PROGRAM SafetyInterface_MtrCntrl052
VAR
	
	pMtrRunning: POINTER TO ConvMtrRunningPuck;
	pSafety: POINTER TO Plc2PlcDataSafetyPuckConv;
	
// Stn052_05_StnMain.MotorCtrl
// Call to motor control function block for each main line motor
// Blue Recv - Enc54: 7, 8, 9  Enc55: 5,6
// Red Recv  - Enc54: 4, 5, 6  Enc55: 3, 4
// Grn Recv  - Enc54: 1, 2, 3  Enc55: 1, 2

	{attribute 'TcLinkToOSO':= '	
		.Enc055Mtr01.iDisconnectOk :=  <0,1,4>TIIB[N31S00 (AL1332)]^N31S05 (AL2341)^TxPDO^input byte 1;
		.Enc055Mtr02.iDisconnectOk :=  <0,1,2>TIIB[N32S00 (AL1332)]^N32S01 (AL2341)^TxPDO^input byte 3;
		.Enc055Mtr03.iDisconnectOk :=  <0,1,4>TIIB[N31S00 (AL1332)]^N31S07 (AL2341)^TxPDO^input byte 3;
		.Enc055Mtr04.iDisconnectOk :=  <0,1,3>TIIB[N32S00 (AL1332)]^N32S01 (AL2341)^TxPDO^input byte 1;
		.Enc055Mtr05.iDisconnectOk :=  <0,1,4>TIIB[N31S00 (AL1332)]^N31S05 (AL2341)^TxPDO^input byte 3;
		.Enc055Mtr06.iDisconnectOk :=  <0,1,3>TIIB[N32S00 (AL1332)]^N32S01 (AL2341)^TxPDO^input byte 3;
		.Enc054Mtr01.iDisconnectOk :=  <0,1,3>TIIB[N26S00 (AL1332)]^N26S04 (AL2341)^TxPDO^input byte 3;
		.Enc054Mtr02.iDisconnectOk :=  <0,1,3>TIIB[N27S00 (AL1332)]^N27S04 (AL2341)^TxPDO^input byte 3;
		.Enc054Mtr03.iDisconnectOk :=  <0,1,3>TIIB[N27S00 (AL1332)]^N27S04 (AL2341)^TxPDO^input byte 3;
		.Enc054Mtr04.iDisconnectOk :=  <0,1,4>TIIB[N26S00 (AL1332)]^N26S04 (AL2341)^TxPDO^input byte 1;
		.Enc054Mtr05.iDisconnectOk :=  <0,1,4>TIIB[N27S00 (AL1332)]^N27S04 (AL2341)^TxPDO^input byte 1;
		.Enc054Mtr06.iDisconnectOk :=  <0,1,4>TIIB[N28S00 (AL1332)]^N28S04 (AL2341)^TxPDO^input byte 1;
		.Enc054Mtr07.iDisconnectOk :=  <0,1,4>TIIB[N26S00 (AL1332)]^N26S04 (AL2341)^TxPDO^input byte 3;
		.Enc054Mtr08.iDisconnectOk :=  <0,1,4>TIIB[N27S00 (AL1332)]^N27S04 (AL2341)^TxPDO^input byte 3;
		.Enc054Mtr09.iDisconnectOk :=  <0,1,4>TIIB[N28S00 (AL1332)]^N28S04 (AL2341)^TxPDO^input byte 3'}
	{attribute 'TcLinkTo':= '	
		.Enc055Mtr01.iOverloadTripped := TIIB[N30S06 (EL1008)]^Channel 6^Input;
		.Enc055Mtr02.iOverloadTripped := TIIB[N30S06 (EL1008)]^Channel 8^Input;
		.Enc055Mtr03.iOverloadTripped := TIIB[N30S07 (EL1008)]^Channel 2^Input;
		.Enc055Mtr04.iOverloadTripped := TIIB[N30S07 (EL1008)]^Channel 4^Input;
		.Enc055Mtr05.iOverloadTripped := TIIB[N30S07 (EL1008)]^Channel 6^Input;
		.Enc055Mtr06.iOverloadTripped := TIIB[N30S07 (EL1008)]^Channel 8^Input;
		.Enc054Mtr01.iOverloadTripped := TIIB[N25S06 (EL1008)]^Channel 6^Input;
		.Enc054Mtr02.iOverloadTripped := TIIB[N25S06 (EL1008)]^Channel 8^Input;
		.Enc054Mtr03.iOverloadTripped := TIIB[N25S07 (EL1008)]^Channel 2^Input;
		.Enc054Mtr04.iOverloadTripped := TIIB[N25S07 (EL1008)]^Channel 4^Input;
		.Enc054Mtr05.iOverloadTripped := TIIB[N25S07 (EL1008)]^Channel 6^Input;
		.Enc054Mtr06.iOverloadTripped := TIIB[N25S07 (EL1008)]^Channel 8^Input;
		.Enc054Mtr07.iOverloadTripped := TIIB[N25S08 (EL1008)]^Channel 2^Input;
		.Enc054Mtr08.iOverloadTripped := TIIB[N25S08 (EL1008)]^Channel 4^Input;
		.Enc054Mtr09.iOverloadTripped := TIIB[N25S08 (EL1008)]^Channel 6^Input;
		.Enc055Mtr01.iRunning := TIIB[N30S06 (EL1008)]^Channel 5^Input;
		.Enc055Mtr02.iRunning := TIIB[N30S06 (EL1008)]^Channel 7^Input;
		.Enc055Mtr03.iRunning := TIIB[N30S07 (EL1008)]^Channel 1^Input;
		.Enc055Mtr04.iRunning := TIIB[N30S07 (EL1008)]^Channel 3^Input;
		.Enc055Mtr05.iRunning := TIIB[N30S07 (EL1008)]^Channel 5^Input;
		.Enc055Mtr06.iRunning := TIIB[N30S07 (EL1008)]^Channel 7^Input;
		.Enc054Mtr01.iRunning := TIIB[N25S06 (EL1008)]^Channel 5^Input;
		.Enc054Mtr02.iRunning := TIIB[N25S06 (EL1008)]^Channel 7^Input;
		.Enc054Mtr03.iRunning := TIIB[N25S07 (EL1008)]^Channel 1^Input;
		.Enc054Mtr04.iRunning := TIIB[N25S07 (EL1008)]^Channel 3^Input;
		.Enc054Mtr05.iRunning := TIIB[N25S07 (EL1008)]^Channel 5^Input;
		.Enc054Mtr06.iRunning := TIIB[N25S07 (EL1008)]^Channel 7^Input;
		.Enc054Mtr07.iRunning := TIIB[N25S08 (EL1008)]^Channel 1^Input;
		.Enc054Mtr08.iRunning := TIIB[N25S08 (EL1008)]^Channel 3^Input;
		.Enc054Mtr09.iRunning := TIIB[N25S08 (EL1008)]^Channel 5^Input;
		.Enc055Mtr01.oRun := TIIB[N30S12 (EL2008)]^Channel 4^Output;
		.Enc055Mtr02.oRun := TIIB[N30S12 (EL2008)]^Channel 5^Output;
		.Enc055Mtr03.oRun := TIIB[N30S12 (EL2008)]^Channel 6^Output;
		.Enc055Mtr04.oRun := TIIB[N30S12 (EL2008)]^Channel 7^Output;
		.Enc055Mtr05.oRun := TIIB[N30S12 (EL2008)]^Channel 8^Output;
		.Enc055Mtr06.oRun := TIIB[N30S13 (EL2008)]^Channel 1^Output;
		.Enc054Mtr01.oRun := TIIB[N25S12 (EL2008)]^Channel 5^Output;
		.Enc054Mtr02.oRun := TIIB[N25S12 (EL2008)]^Channel 6^Output;
		.Enc054Mtr03.oRun := TIIB[N25S12 (EL2008)]^Channel 7^Output;
		.Enc054Mtr04.oRun := TIIB[N25S12 (EL2008)]^Channel 8^Output;
		.Enc054Mtr05.oRun := TIIB[N25S13 (EL2008)]^Channel 1^Output;
		.Enc054Mtr06.oRun := TIIB[N25S13 (EL2008)]^Channel 2^Output;
		.Enc054Mtr07.oRun := TIIB[N25S13 (EL2008)]^Channel 3^Output;
		.Enc054Mtr08.oRun := TIIB[N25S13 (EL2008)]^Channel 4^Output;
		.Enc054Mtr09.oRun := TIIB[N25S13 (EL2008)]^Channel 5^Output'}
	MtrCtrls: ConvMtrCtrlsPuck;

	MtrNOKtoRun : BOOL;	
	cntMotorStartIndex: DINT;	
	tmrMotorStartIndex: TON;


END_VAR
VAR CONSTANT	
	
	cMaxMotorStartIndex :DINT := 9;  //If starting pairs of motors  adjust to max number of motors "per enclosure" /2
	
END_VAR

pMtrRunning := ADR(gProduced_SafetyInterfaceConv.MtrRunning);
pSafety := ADR(gProduced_SafetyInterfaceConv);

//Create sequenced motor start index - to prevent inrush overloads at time of motor start		
tmrMotorStartIndex(IN:=NOT tmrMotorStartIndex.Q,PT:=T#300ms);		
IF tmrMotorStartIndex.Q THEN 		
	cntMotorStartIndex := cntMotorStartIndex + 1;	
	IF cntMotorStartIndex > cMaxMotorStartIndex THEN 	
		cntMotorStartIndex := 1;
	END_IF	
END_IF		

// Call action code block that does call for each main line motor		
MotorCtrl();

//distibute the incoming stn data (consumed data from stn) to single produced outgoing to all stns
//MEMCPY(ADR(gProduced_SafetyInterfaceConv.gMtrRunningStn051), ADR(gMtrRunning), SizeOf(gProduced_SafetyInterfaceConv.gMtrRunningStn051));

ACTION MotorCtrl:
// Stn052_05_StnMain.MotorCtrl
// Call to motor control function block for each main line motor
// Blue Recv - Enc54: 7, 8, 9  Enc55: 5,6
// Red Recv  - Enc54: 4, 5, 6  Enc55: 3, 4
// Grn Recv  - Enc54: 1, 2, 3  Enc55: 1, 2
MtrCtrls.Enc054Mtr01(
	CycleAuto := gConsumed_Stn052ToSafetyInterface.CycleAuto,
	CycleReset := gConsumed_Stn052ToSafetyInterface.CycleReset,
	NOKtoRun := pSafety^.Enc054.iEstopRlyTripped,	
//	NOKtoRun := pSafety^.Enc054.iEstopRlyTripped OR 
//		NOT gConsumed_Stn052ToSafetyInterface.Stn052PLCData[2].3 OR 
//		NOT gConsumed_Stn052ToSafetyInterface_OK,		
	StartIndexThisMotor := 1,
	StartIndexCurrent := cntMotorStartIndex,
	hoMtrName := 'Enc054-Mtr1',
	MtrRunning => pMtrRunning^.Enc054Mtr01);

MtrCtrls.Enc054Mtr02(	
	CycleAuto := gConsumed_Stn052ToSafetyInterface.CycleAuto,
	CycleReset := gConsumed_Stn052ToSafetyInterface.CycleReset,
	NOKtoRun := pSafety^.Enc054.iEstopRlyTripped,	
//	NOKtoRun := pSafety^.Enc054.iEstopRlyTripped OR 
//		NOT gConsumed_Stn052ToSafetyInterface.Stn052PLCData[2].3 OR 
//		NOT gConsumed_Stn052ToSafetyInterface_OK,		
	StartIndexThisMotor := 1,
	StartIndexCurrent := cntMotorStartIndex,
	hoMtrName := 'Enc054-Mtr2',
	MtrRunning => pMtrRunning^.Enc054Mtr02);

MtrCtrls.Enc054Mtr03(	
	CycleAuto := gConsumed_Stn052ToSafetyInterface.CycleAuto,
	CycleReset := gConsumed_Stn052ToSafetyInterface.CycleReset,
	NOKtoRun := pSafety^.Enc054.iEstopRlyTripped,	
//	NOKtoRun := pSafety^.Enc054.iEstopRlyTripped OR 
//		NOT gConsumed_Stn052ToSafetyInterface.Stn052PLCData[2].3 OR 
//		NOT gConsumed_Stn052ToSafetyInterface_OK,		
	StartIndexThisMotor := 2,
	StartIndexCurrent := cntMotorStartIndex,
	hoMtrName := 'Enc054-Mtr3',
	MtrRunning => pMtrRunning^.Enc054Mtr03);

MtrCtrls.Enc054Mtr04(	
	CycleAuto := gConsumed_Stn052ToSafetyInterface.CycleAuto,
	CycleReset := gConsumed_Stn052ToSafetyInterface.CycleReset,
	NOKtoRun := pSafety^.Enc054.iEstopRlyTripped,	
//	NOKtoRun := pSafety^.Enc054.iEstopRlyTripped OR 
//		NOT gConsumed_Stn052ToSafetyInterface.Stn052PLCData[2].3 OR 
//		NOT gConsumed_Stn052ToSafetyInterface_OK,		
	StartIndexThisMotor := 2,
	StartIndexCurrent := cntMotorStartIndex,
	hoMtrName := 'Enc054-Mtr4',
	MtrRunning => pMtrRunning^.Enc054Mtr04);

MtrCtrls.Enc054Mtr05(	
	CycleAuto := gConsumed_Stn052ToSafetyInterface.CycleAuto,
	CycleReset := gConsumed_Stn052ToSafetyInterface.CycleReset,
	NOKtoRun := pSafety^.Enc054.iEstopRlyTripped,	
//	NOKtoRun := pSafety^.Enc054.iEstopRlyTripped OR 
//		NOT gConsumed_Stn052ToSafetyInterface.Stn052PLCData[2].3 OR 
//		NOT gConsumed_Stn052ToSafetyInterface_OK,		
	StartIndexThisMotor := 3,
	StartIndexCurrent := cntMotorStartIndex,
	hoMtrName := 'Enc054-Mtr5',
	MtrRunning => pMtrRunning^.Enc054Mtr05);

MtrCtrls.Enc054Mtr06(	
	CycleAuto := gConsumed_Stn052ToSafetyInterface.CycleAuto,
	CycleReset := gConsumed_Stn052ToSafetyInterface.CycleReset,
	NOKtoRun := pSafety^.Enc054.iEstopRlyTripped,	
//	NOKtoRun := pSafety^.Enc054.iEstopRlyTripped OR 
//		NOT gConsumed_Stn052ToSafetyInterface.Stn052PLCData[2].3 OR 
//		NOT gConsumed_Stn052ToSafetyInterface_OK,		
	StartIndexThisMotor := 3,
	StartIndexCurrent := cntMotorStartIndex,
	hoMtrName := 'Enc054-Mtr6',
	MtrRunning => pMtrRunning^.Enc054Mtr06);

MtrCtrls.Enc054Mtr07(	
	CycleAuto := gConsumed_Stn052ToSafetyInterface.CycleAuto,
	CycleReset := gConsumed_Stn052ToSafetyInterface.CycleReset,
	NOKtoRun := pSafety^.Enc054.iEstopRlyTripped,	
//	NOKtoRun := pSafety^.Enc054.iEstopRlyTripped OR 
//		NOT gConsumed_Stn052ToSafetyInterface.Stn052PLCData[2].3 OR 
//		NOT gConsumed_Stn052ToSafetyInterface_OK,		
	StartIndexThisMotor := 4,
	StartIndexCurrent := cntMotorStartIndex,
	hoMtrName := 'Enc054-Mtr7',
	MtrRunning => pMtrRunning^.Enc054Mtr07);

MtrCtrls.Enc054Mtr08(	
	CycleAuto := gConsumed_Stn052ToSafetyInterface.CycleAuto,
	CycleReset := gConsumed_Stn052ToSafetyInterface.CycleReset,
	NOKtoRun := pSafety^.Enc054.iEstopRlyTripped,	
//	NOKtoRun := pSafety^.Enc054.iEstopRlyTripped OR 
//		NOT gConsumed_Stn052ToSafetyInterface.Stn052PLCData[2].3 OR 
//		NOT gConsumed_Stn052ToSafetyInterface_OK,		
	StartIndexThisMotor := 4,
	StartIndexCurrent := cntMotorStartIndex,
	hoMtrName := 'Enc054-Mtr8',
	MtrRunning => pMtrRunning^.Enc054Mtr08);

MtrCtrls.Enc054Mtr09(	
	CycleAuto := gConsumed_Stn052ToSafetyInterface.CycleAuto,
	CycleReset := gConsumed_Stn052ToSafetyInterface.CycleReset,
	NOKtoRun := pSafety^.Enc054.iEstopRlyTripped,	
//	NOKtoRun := pSafety^.Enc054.iEstopRlyTripped OR 
//		NOT gConsumed_Stn052ToSafetyInterface.Stn052PLCData[2].3 OR 
//		NOT gConsumed_Stn052ToSafetyInterface_OK,		
	StartIndexThisMotor := 5,
	StartIndexCurrent := cntMotorStartIndex,
	hoMtrName := 'Enc054-Mtr9',
	MtrRunning => pMtrRunning^.Enc054Mtr09);

MtrCtrls.Enc055Mtr01(	
	CycleAuto := gConsumed_Stn052ToSafetyInterface.CycleAuto,
	CycleReset := gConsumed_Stn052ToSafetyInterface.CycleReset,
	NOKtoRun := pSafety^.Enc055.iEstopRlyTripped,	
//	NOKtoRun := pSafety^.Enc055.iEstopRlyTripped OR 
//		NOT gConsumed_Stn052ToSafetyInterface.Stn052PLCData[2].3 OR 
//		NOT gConsumed_Stn052ToSafetyInterface_OK,		
	StartIndexThisMotor := 1,
	StartIndexCurrent := cntMotorStartIndex,
	hoMtrName := 'Enc055-Mtr1',
	MtrRunning => pMtrRunning^.Enc055Mtr01);

MtrCtrls.Enc055Mtr02(	
	CycleAuto := gConsumed_Stn052ToSafetyInterface.CycleAuto,
	CycleReset := gConsumed_Stn052ToSafetyInterface.CycleReset,
	NOKtoRun := pSafety^.Enc055.iEstopRlyTripped,	
//	NOKtoRun := pSafety^.Enc055.iEstopRlyTripped OR 
//		NOT gConsumed_Stn052ToSafetyInterface.Stn052PLCData[2].3 OR 
//		NOT gConsumed_Stn052ToSafetyInterface_OK,		
	StartIndexThisMotor := 1,
	StartIndexCurrent := cntMotorStartIndex,
	hoMtrName := 'Enc055-Mtr2',
	MtrRunning => pMtrRunning^.Enc055Mtr02);

MtrCtrls.Enc055Mtr03(	
	CycleAuto := gConsumed_Stn052ToSafetyInterface.CycleAuto,
	CycleReset := gConsumed_Stn052ToSafetyInterface.CycleReset,
	NOKtoRun := pSafety^.Enc055.iEstopRlyTripped,	
//	NOKtoRun := pSafety^.Enc055.iEstopRlyTripped OR 
//		NOT gConsumed_Stn052ToSafetyInterface.Stn052PLCData[2].3 OR 
//		NOT gConsumed_Stn052ToSafetyInterface_OK,		
	StartIndexThisMotor := 2,
	StartIndexCurrent := cntMotorStartIndex,
	hoMtrName := 'Enc055-Mtr3',
	MtrRunning => pMtrRunning^.Enc055Mtr03);

MtrCtrls.Enc055Mtr04(	
	CycleAuto := gConsumed_Stn052ToSafetyInterface.CycleAuto,
	CycleReset := gConsumed_Stn052ToSafetyInterface.CycleReset,
	NOKtoRun := pSafety^.Enc055.iEstopRlyTripped,	
//	NOKtoRun := pSafety^.Enc055.iEstopRlyTripped OR 
//		NOT gConsumed_Stn052ToSafetyInterface.Stn052PLCData[2].3 OR 
//		NOT gConsumed_Stn052ToSafetyInterface_OK,		
	StartIndexThisMotor := 2,
	StartIndexCurrent := cntMotorStartIndex,
	hoMtrName := 'Enc055-Mtr4',
	MtrRunning => pMtrRunning^.Enc055Mtr04);

MtrCtrls.Enc055Mtr05(	
	CycleAuto := gConsumed_Stn052ToSafetyInterface.CycleAuto,
	CycleReset := gConsumed_Stn052ToSafetyInterface.CycleReset,
	NOKtoRun := pSafety^.Enc055.iEstopRlyTripped,	
//	NOKtoRun := pSafety^.Enc055.iEstopRlyTripped OR 
//		NOT gConsumed_Stn052ToSafetyInterface.Stn052PLCData[2].3 OR 
//		NOT gConsumed_Stn052ToSafetyInterface_OK,		
	StartIndexThisMotor := 3,
	StartIndexCurrent := cntMotorStartIndex,
	hoMtrName := 'Enc055-Mtr5',
	MtrRunning => pMtrRunning^.Enc055Mtr05);

MtrCtrls.Enc055Mtr06(	
	CycleAuto := gConsumed_Stn052ToSafetyInterface.CycleAuto,
	CycleReset := gConsumed_Stn052ToSafetyInterface.CycleReset,
	NOKtoRun := pSafety^.Enc055.iEstopRlyTripped,	
//	NOKtoRun := pSafety^.Enc055.iEstopRlyTripped OR 
//		NOT gConsumed_Stn052ToSafetyInterface.Stn052PLCData[2].3 OR 
//		NOT gConsumed_Stn052ToSafetyInterface_OK,		
	StartIndexThisMotor := 3,
	StartIndexCurrent := cntMotorStartIndex,
	hoMtrName := 'Enc055-Mtr6',
	MtrRunning => pMtrRunning^.Enc055Mtr06);


	
//For each motor that the station needs running information but NOT actually controlling the output… 
//(populate the running bit from the produced consumed logic)

// Populate motor running for motors controlled (outputs linked) by other stations
//gMtrRunning.Enc062Mtr07 := gConsumed_Stn901To902.ScratchPad[10].0;
END_ACTION

END_PROGRAM

(* stored: Version 1.1.0.1, ProductVersion 3.1.4024.6
   POU SafetyInterface_MtrCntrl052: Id {b45e1794-8829-4c37-b1bb-5bde821ec8d0}, SpecialFunc None
   Action MotorCtrl: Id {5a40751f-d445-43e6-9651-238ae7e18c2e} *)
